(* unknown state *)
ELSE

	eState := E_TCPIP_IDLE;

	(* clear outputs *)
	bDone := FALSE;
	bBusy := FALSE;
	bError := FALSE;
	nErrorID := 0;
END_CASE

END_FUNCTION_BLOCK

// ---- POUs/SOFTWARE_lib/TCP FBs/FB_TCP_ReceiveData_V2.TcPOU
(* poll TCP Server for incoming data *)
FUNCTION_BLOCK FB_TCP_ReceiveData_V2
VAR_INPUT
	bEnable				: BOOL;			(* set TRUE to enable periodic TCP data receive *)
	hSocket				: T_HSocket;	(* TCP socket *)
	tUpdateTime			: TIME;			(* receive update rate *)
END_VAR
VAR_IN_OUT
	strTCPData			: T_MaxString;	(* string to which incoming TCP data will be appended *)
END_VAR
VAR_OUTPUT
	bDone				: BOOL;			(* TRUE = TCP receive done *)
	bBusy				: BOOL;			(* TRUE = TCP receive in progress *)
	bError				: BOOL;			(* TRUE = TCP receive error *)
	nErrorID			: UDINT;		(* TCP receive error code *)
	bDataReceived		: BOOL;			(* TRUE = data received *)
END_VAR
VAR
	fbTimer				: TON;
	eState				: E_TCPIP_State;
	fbTCPReceive		: FB_SocketReceive;
	strTCPRxChars		: T_MaxString;
END_VAR
(*
-------------------------------------------------------------------------------------------------
Date		Version	Author	Comments
-------------------------------------------------------------------------------------------------
16/08/2012	1.40.02	PB		Initial release

-------------------------------------------------------------------------------------------------
*)

(* TCP receive timer *)
fbTimer(
	IN	:= bEnable,
	PT	:= tUpdateTime
);

CASE eState OF

	(* idle state *)
	E_TCPIP_IDLE:

		(* receive data *)
		IF fbTimer.Q = TRUE THEN

			(* reset TCP receive timer *)
			fbTimer(IN := FALSE);

			(* update status outputs *)
			bDone := FALSE;
			bBusy := TRUE;
			bError := FALSE;
			nErrorID := 0;
			bDataReceived := FALSE;

			(* clear TCP receive string *)
			MEMSET(ADR(strTCPRxChars), 16#00, SIZEOF(strTCPRxChars));

			eState := E_TCPIP_RECEIVE;

		(* no action required *)
		ELSE

			bDone := FALSE;
			bBusy := FALSE;
			bError := FALSE;
			nErrorID := 0;
			bDataReceived := FALSE;
		END_IF


	(* receive data *)
	E_TCPIP_RECEIVE:

		(* receive data from TCP server *)
		fbTCPReceive(
			sSrvNetId	:= '',
			hSocket		:= hSocket,
			cbLen		:= SIZEOF(strTCPRxChars),
			pDest		:= ADR(strTCPRxChars),
			bExecute	:= TRUE,
			tTimeout	:= T#500ms
		);
		
		(* receive TCP data complete *)
		IF fbTCPReceive.bBusy = FALSE THEN
		
			(* receive TCP data completed OK *)
			IF fbTCPReceive.bError = FALSE THEN

				(* 1 or more data bytes received *)
				IF fbTCPReceive.nRecBytes > 0 THEN

					(* append returned data to TCP data string *)
					strTCPData := CONCAT(strTCPData, strTCPRxChars);
					bDataReceived := TRUE;

				(* no data received *)
				ELSE

					bDataReceived := FALSE;
				END_IF

			(* receive data error *)
			ELSE

				bError := TRUE;
				nErrorID := fbTCPReceive.nErrId;
			END_IF
		
			eState :=E_TCPIP_DONE;

			(* close off fbReceiveTCPData *)
			fbTCPReceive(bExecute := FALSE);
		END_IF


	(* done *)
	E_TCPIP_DONE:

		bDone := TRUE;
		bBusy := FALSE;

		eState :=E_TCPIP_IDLE;


	(* unknown state *)
	ELSE

		(* close off FBs *)
		fbTCPReceive(bExecute := FALSE);
		fbTimer(IN := FALSE);

		eState :=E_TCPIP_IDLE;

END_CASE

END_FUNCTION_BLOCK

// ---- POUs/SOFTWARE_lib/TCP FBs/FB_TCP_SendData.TcPOU
(* send data to TCP socket *)
FUNCTION_BLOCK FB_TCP_SendData
VAR_INPUT
	bExecute		: BOOL;			(* set TRUE to send data to TCP socket *)
	hSocket			: T_HSocket;	(* TCP socket handle *)
	pDataAdr		: POINTER TO BYTE;	(* pointer to data to send to TCP port *)
	nDataBytes		: UDINT;		(* number of bytes to send to TCP port *)
	tTimeout		: TIME;			(* TCP timeout *)
END_VAR
VAR_OUTPUT
	bDone			: BOOL;			(* TRUE = command complete *)
	bBusy			: BOOL;			(* TRUE = command in progress *)
	bError			: BOOL;			(* TRUE = error occurred with command *)
	nErrorID		: UDINT;		(* error code *)
END_VAR
VAR
	fbExecute		: R_TRIG;
	eState			: E_TCPIP_State;
	fbSendCommand	: FB_SocketSend;
END_VAR
(*
-------------------------------------------------------------------------------------------------
Date		Version	Author	Comments
-------------------------------------------------------------------------------------------------
			2.00.00	PB		Initial release

-------------------------------------------------------------------------------------------------
*)

(* compare files on rising edge of bExecute *)
fbExecute(CLK := bExecute);

CASE eState OF

	(* idle state *)
	E_TCPIP_IDLE:

		(* start new cycle *)
		IF fbExecute.Q = TRUE THEN

			(* reset status outputs *)
			bDone := FALSE;
			bBusy := TRUE;
			bError := FALSE;
			nErrorID := 0;

			eState := E_TCPIP_SEND;

		(* reset status outputs when bExecute is reset *)
		ELSIF bExecute = FALSE THEN

			bDone := FALSE;
			bBusy := FALSE;
			bError := FALSE;
			nErrorID := 0;
		END_IF


	(* send command *)
	E_TCPIP_SEND:

		(* send command *)
		fbSendCommand(
			sSrvNetId	:= '',
			hSocket		:= hSocket,
			cbLen		:= nDataBytes,
			pSrc		:= pDataAdr,
			bExecute	:= TRUE,
			tTimeout	:= T#1s,
		);

		(* send command complete *)
		IF fbSendCommand.bBusy = FALSE THEN

			(* send command completed OK *)
			IF fbSendCommand.bError = FALSE THEN

				eState := E_TCPIP_DONE;

			(* send command error *)
			ELSE

				bError := TRUE;
				nErrorID := fbSendCommand.nErrId;

				eState := E_TCPIP_DONE;
			END_IF

			(* close off fbSendCommand *)
			fbSendCommand(bExecute := FALSE);
		END_IF


	(* TCP command done *)
	E_TCPIP_DONE:

		bBusy := FALSE;
		bDone := TRUE;

		eState := E_TCPIP_IDLE;

(* unknown state *)
ELSE

	eState := E_TCPIP_IDLE;
END_CASE

END_FUNCTION_BLOCK

// ---- POUs/SOFTWARE_lib/TCP FBs/FB_TCP_ServerPortCtrl.TcPOU
(* TCP port ctrl for Server-Client devices *)
FUNCTION_BLOCK FB_TCP_ServerPortCtrl
VAR_INPUT
	bEnable				: BOOL;			(* set TRUE to enable TCP connection *)
	eMode				: E_SocketAcceptMode;	(* specifies which connections to accept *)
	strRemoteIPAddr		: T_IPv4Addr;	(* IP address for remote device *)
	strLocalIPAddr		: T_IPv4Addr;	(* IP address for local device *)
	nLocalPortNo		: UINT;			(* port number for local device *)
	tReconnectTime		: TIME;			(* TCP reconnect time *)
END_VAR
VAR_OUTPUT
	bConnected			: BOOL;			(* TRUE = TCP port is currently open *)
	bError				: BOOL;			(* TRUE = error occurred when opening TCP port *)
	nErrorID			: UDINT;		(* TRUE = error code *)
	hSocket				: T_HSocket;	(* TCP socket handle *)
	nSyncOffset			: DINT;			(* sync offset value to spread TCP Server access load *)
	eSocketState		: E_SocketConnectionState;	(* TCP socket state *)
END_VAR
VAR
	strTargetIPAddr		: T_IPv4Addr;
	arrTargetIPAddr		: T_IPv4AddrArr;
	nTargetPortNo		: UDINT;
	eTCPState			: E_TCPIP_State;
	bServerHndOK		: BOOL;
	hServer				: T_HSERVER;
	fbTCPPortCtrl		: FB_ServerClientConnection;
END_VAR
(*
-------------------------------------------------------------------------------------------------
Date		Version	Author	Comments
-------------------------------------------------------------------------------------------------
30/01/2015	3.00.00	PB		nRemotePort input removed as it is not used

-------------------------------------------------------------------------------------------------
06/09/2012	1.41.00	PB		FB now re-connects properly if strRemoteIPAddr or nRemotePortNo are changed while TCP connection is active.
							bError and nErrorID now linked directly to FB_ServerClientConnection.
22/11/2011	1.34.00	PB		Initial release.

-------------------------------------------------------------------------------------------------
*)

CASE eTCPState OF

	(* TCP connetion not active *)
	E_TCPIP_IDLE:

		(* TCP connection is enabled *)
		IF bEnable = TRUE THEN

			(* target IP address and port number *)
			strTargetIPAddr := strRemoteIPAddr;
			nTargetPortNo := nLocalPortNo;

			(* convert target IP address to bytes *)
			arrTargetIPAddr := F_ScanIPv4AddrIds(strTargetIPAddr);
			nSyncOffset := arrTargetIPAddr[3] MOD 10;

			eTCPState := E_TCPIP_CONNECT;
		END_IF


	(* open TCP connection *)
	E_TCPIP_CONNECT:

		(* close TCP connection *)
		IF bEnable = FALSE THEN

			eTCPState := E_TCPIP_DISCONNECT;

		(* TCP connect error or remote IP address or local port number have changed while connection is active *)
		ELSIF fbTCPPortCtrl.bError = TRUE OR (strRemoteIPAddr <> strTargetIPAddr AND strRemoteIPAddr <> '') OR (nLocalPortNo <> nTargetPortNo AND nLocalPortNo <> 0) THEN

			eTCPState := E_TCPIP_DISCONNECT;
		END_IF


	(* close TCP connection *)
	E_TCPIP_DISCONNECT:

		(* TCP port has been closed *)
		IF eSocketState = eSOCKET_DISCONNECTED THEN

			eTCPState := E_TCPIP_IDLE;
		END_IF


(* unknown state *)
ELSE

	eTCPState := E_TCPIP_IDLE;
END_CASE

(* create local server handle *)
bServerHndOK := F_CreateServerHnd('', strLocalIPAddr, nTargetPortNo, LISTEN_MODE_CLOSEALL(* OR CONNECT_MODE_ENABLEDBG*), FALSE, hServer);


(* TCP port connection ctrl *)
fbTCPPortCtrl(
	eMode		:= eMode,
	sRemoteHost	:= strTargetIPAddr,
	nRemotePort	:= nTargetPortNo,
	bEnable		:= bServerHndOK AND eTCPState = E_TCPIP_CONNECT,
	tReconnect	:= tReconnectTime,
	hServer		:= hServer,
	bError		=> bError,
	nErrID		=> nErrorID,
	hSocket		=> hSocket,
	eState		=> eSocketState
);

(* connected status *)
bConnected := eSocketState = eSOCKET_CONNECTED;

END_FUNCTION_BLOCK

// ---- POUs/Tests/FB_FIND_OuterDuplicates.TcPOU
FUNCTION_BLOCK FB_FIND_OuterDuplicates
VAR_INPUT
END_VAR
VAR_OUTPUT
	bHasDuplicates		: BOOL;
	nDuplicateCount		: UINT;
	nIterationCount		: UINT;
END_VAR
VAR
	nOuterIndex			: UINT;
	nMax_Outers			: UINT := 50;
	nMax_Packs			: UINT := 10;
	nInnerOuterIndex	: UINT;
	nInnerPackIndex		: UINT;
	nPackIndex			: UINT;
	sCurrentOuterCode	: T_MaxString;
	sCurrentPackCode	: T_MaxString;	
	bIsDuplicate 		: BOOL;
	bISOuterDuplicate	: BOOL;
END_VAR
VAR_IN_OUT	
	stCase				: ST_LAB_CaseData;
END_VAR


bHasDuplicates := FALSE;
nDuplicateCount := 0;
	
	(* Loop throught all packs in one case 'stCase' *)
	FOR nOuterIndex := 1 TO nMax_Outers DO
		sCurrentOuterCode := stCase.aOuters[nOuterIndex].sOuterCode;
		FOR nPackIndex := 1 TO nMax_Packs DO
			sCurrentPackCode := stCase.aOuters[nOuterIndex].aPacks[nPackIndex].sPackCode;
			bIsDuplicate := FALSE;			
			(* Looking for same pack codes in all outers *)
			FOR nInnerOuterIndex := nOuterIndex TO nMax_Outers DO
				IF nInnerOuterIndex < 50 THEN					
					IF (sCurrentOuterCode = stCase.aOuters[nInnerOuterIndex + 1].sOuterCode) THEN
						bIsOuterDuplicate									:= TRUE;													
						stCase.aOuters[nOuterIndex].nOuterRejectID			:= 200;					
						stCase.aOuters[nInnerOuterIndex + 1].nOuterRejectID	:= 200;
					END_IF	
				END_IF
				FOR nInnerPackIndex := 1 TO nMax_Packs DO
					nIterationCount	:= nIterationCount + 1;					
					(* Exclude comparing same pack with itself *)
					IF NOT ((nInnerOuterIndex = nOuterIndex) AND (nInnerPackIndex = nPackIndex)) THEN
						IF sCurrentPackCode = stCase.aOuters[nInnerOuterIndex].aPacks[nInnerPackIndex].sPackCode THEN
							bIsDuplicate := TRUE;
							nDuplicateCount := nDuplicateCount + 1;
							
							stCase.aOuters[nInnerOuterIndex].aPacks[nInnerPackIndex].nPackRejectID	:= 200;
							stCase.aOuters[nInnerOuterIndex].nOuterRejectID							:= 200;
							
							stCase.aOuters[nOuterIndex].aPacks[nPackIndex].nPackRejectID			:= 200;
							stCase.aOuters[nOuterIndex].nOuterRejectID								:= 200;
						END_IF
					END_IF
				END_FOR
			END_FOR			
			IF bIsDuplicate THEN
				bHasDuplicates 	:= TRUE;
			END_IF
		END_FOR
	END_FOR
	
	
	(* nDuplicateCount includes all elements with same pack codes *)
	(* the number of duplicated codes is nDuplicateCount/2 *)

END_FUNCTION_BLOCK

// ---- POUs/Tests/Outer_IN_Case_Duplicat.TcPOU
PROGRAM Outer_IN_Case_Duplicat
VAR
		
	fbFIND_OuterDuplicates		: FB_FIND_OuterDuplicates;
	
	bHasDuplicates				: BOOL;
	nDuplicateCount				: UINT;
	
	rTrig						: R_TRIG;
	bExecute					: BOOL;
	
	
	// dla petli for dla stworzenia outerow 
	rTrigDataFill	: R_TRIG;
	bDataFill		: BOOL;
	
	iOuter		: UINT;
	iPack		: UINT;
	
	sPackNum	: STRING;
	sOuterNum	: STRING;
	sPackCode	: STRING;
	
END_VAR


//CaseDataAdd();
//Case50outersADD();

FullFilOuter();

rTrig(CLK := bExecute);

IF rTrig.Q THEN	
	fbFIND_OuterDuplicates(
		stCase 			:= GVL_test.stCaseFull, 
		bHasDuplicates 	=> bHasDuplicates, 
		nDuplicateCount => nDuplicateCount
	);	
	
END_IF

ACTION Case50outersADD:
(* ===== OUTER 1 ===== *)
GVL_test.stCase.aOuters[1].sOuterCode    := 'OUTER1';
GVL_test.stCase.aOuters[1].nOutersStatus := 5;
// packs 1..10
GVL_test.stCase.aOuters[1].aPacks[1].sPackCode   := 'PACK01OUTER1';
GVL_test.stCase.aOuters[1].aPacks[1].nPackStatus := 5;
GVL_test.stCase.aOuters[1].aPacks[2].sPackCode   := 'PACK02OUTER1';
GVL_test.stCase.aOuters[1].aPacks[2].nPackStatus := 5;
GVL_test.stCase.aOuters[1].aPacks[3].sPackCode   := 'PACK03OUTER1';
GVL_test.stCase.aOuters[1].aPacks[3].nPackStatus := 5;
GVL_test.stCase.aOuters[1].aPacks[4].sPackCode   := 'PACK04OUTER1';
GVL_test.stCase.aOuters[1].aPacks[4].nPackStatus := 5;
GVL_test.stCase.aOuters[1].aPacks[5].sPackCode   := 'PACK05OUTER1';
GVL_test.stCase.aOuters[1].aPacks[5].nPackStatus := 5;
GVL_test.stCase.aOuters[1].aPacks[6].sPackCode   := 'PACK06OUTER1';
GVL_test.stCase.aOuters[1].aPacks[6].nPackStatus := 5;
GVL_test.stCase.aOuters[1].aPacks[7].sPackCode   := 'PACK07OUTER1';
GVL_test.stCase.aOuters[1].aPacks[7].nPackStatus := 5;
GVL_test.stCase.aOuters[1].aPacks[8].sPackCode   := 'PACK08OUTER1';
GVL_test.stCase.aOuters[1].aPacks[8].nPackStatus := 5;
GVL_test.stCase.aOuters[1].aPacks[9].sPackCode   := 'PACK09OUTER1';
GVL_test.stCase.aOuters[1].aPacks[9].nPackStatus := 5;
GVL_test.stCase.aOuters[1].aPacks[10].sPackCode  := 'PACK10OUTER1';
GVL_test.stCase.aOuters[1].aPacks[10].nPackStatus := 5;

(* ===== OUTER 2 ===== *)
GVL_test.stCase.aOuters[2].sOuterCode    := 'OUTER2';
GVL_test.stCase.aOuters[2].nOutersStatus := 5;
// packs 1..10
GVL_test.stCase.aOuters[2].aPacks[1].sPackCode   := 'PACK01OUTER2';
GVL_test.stCase.aOuters[2].aPacks[1].nPackStatus := 5;
GVL_test.stCase.aOuters[2].aPacks[2].sPackCode   := 'PACK02OUTER2';
GVL_test.stCase.aOuters[2].aPacks[2].nPackStatus := 5;
GVL_test.stCase.aOuters[2].aPacks[3].sPackCode   := 'PACK03OUTER2';
GVL_test.stCase.aOuters[2].aPacks[3].nPackStatus := 5;
GVL_test.stCase.aOuters[2].aPacks[4].sPackCode   := 'PACK04OUTER2';
GVL_test.stCase.aOuters[2].aPacks[4].nPackStatus := 5;
GVL_test.stCase.aOuters[2].aPacks[5].sPackCode   := 'PACK05OUTER2';
GVL_test.stCase.aOuters[2].aPacks[5].nPackStatus := 5;
GVL_test.stCase.aOuters[2].aPacks[6].sPackCode   := 'PACK06OUTER2';
GVL_test.stCase.aOuters[2].aPacks[6].nPackStatus := 5;
GVL_test.stCase.aOuters[2].aPacks[7].sPackCode   := 'PACK07OUTER2';
GVL_test.stCase.aOuters[2].aPacks[7].nPackStatus := 5;
GVL_test.stCase.aOuters[2].aPacks[8].sPackCode   := 'PACK08OUTER2';
GVL_test.stCase.aOuters[2].aPacks[8].nPackStatus := 5;
GVL_test.stCase.aOuters[2].aPacks[9].sPackCode   := 'PACK09OUTER2';
GVL_test.stCase.aOuters[2].aPacks[9].nPackStatus := 5;
GVL_test.stCase.aOuters[2].aPacks[10].sPackCode  := 'PACK10OUTER2';
GVL_test.stCase.aOuters[2].aPacks[10].nPackStatus := 5;

(* ===== OUTER 3 ===== *)
GVL_test.stCase.aOuters[3].sOuterCode    := 'OUTER3';
GVL_test.stCase.aOuters[3].nOutersStatus := 5;
// packs 1..10
GVL_test.stCase.aOuters[3].aPacks[1].sPackCode   := 'PACK01OUTER3';
GVL_test.stCase.aOuters[3].aPacks[1].nPackStatus := 5;
GVL_test.stCase.aOuters[3].aPacks[2].sPackCode   := 'PACK02OUTER3';
GVL_test.stCase.aOuters[3].aPacks[2].nPackStatus := 5;
GVL_test.stCase.aOuters[3].aPacks[3].sPackCode   := 'PACK03OUTER3';
GVL_test.stCase.aOuters[3].aPacks[3].nPackStatus := 5;
GVL_test.stCase.aOuters[3].aPacks[4].sPackCode   := 'PACK04OUTER3';
GVL_test.stCase.aOuters[3].aPacks[4].nPackStatus := 5;
GVL_test.stCase.aOuters[3].aPacks[5].sPackCode   := 'PACK05OUTER3';
GVL_test.stCase.aOuters[3].aPacks[5].nPackStatus := 5;
GVL_test.stCase.aOuters[3].aPacks[6].sPackCode   := 'PACK06OUTER3';
GVL_test.stCase.aOuters[3].aPacks[6].nPackStatus := 5;
GVL_test.stCase.aOuters[3].aPacks[7].sPackCode   := 'PACK07OUTER3';
GVL_test.stCase.aOuters[3].aPacks[7].nPackStatus := 5;
GVL_test.stCase.aOuters[3].aPacks[8].sPackCode   := 'PACK08OUTER3';
GVL_test.stCase.aOuters[3].aPacks[8].nPackStatus := 5;
GVL_test.stCase.aOuters[3].aPacks[9].sPackCode   := 'PACK09OUTER3';
GVL_test.stCase.aOuters[3].aPacks[9].nPackStatus := 5;
GVL_test.stCase.aOuters[3].aPacks[10].sPackCode  := 'PACK10OUTER3';
GVL_test.stCase.aOuters[3].aPacks[10].nPackStatus := 5;

(* ===== OUTER 4 ===== *)
GVL_test.stCase.aOuters[4].sOuterCode    := 'OUTER4';
GVL_test.stCase.aOuters[4].nOutersStatus := 5;
// packs 1..10
GVL_test.stCase.aOuters[4].aPacks[1].sPackCode   := 'PACK01OUTER4';
GVL_test.stCase.aOuters[4].aPacks[1].nPackStatus := 5;
GVL_test.stCase.aOuters[4].aPacks[2].sPackCode   := 'PACK02OUTER4';
GVL_test.stCase.aOuters[4].aPacks[2].nPackStatus := 5;
GVL_test.stCase.aOuters[4].aPacks[3].sPackCode   := 'PACK03OUTER4';
GVL_test.stCase.aOuters[4].aPacks[3].nPackStatus := 5;
GVL_test.stCase.aOuters[4].aPacks[4].sPackCode   := 'PACK04OUTER4';
GVL_test.stCase.aOuters[4].aPacks[4].nPackStatus := 5;
GVL_test.stCase.aOuters[4].aPacks[5].sPackCode   := 'PACK05OUTER4';
GVL_test.stCase.aOuters[4].aPacks[5].nPackStatus := 5;
GVL_test.stCase.aOuters[4].aPacks[6].sPackCode   := 'PACK06OUTER4';
GVL_test.stCase.aOuters[4].aPacks[6].nPackStatus := 5;
GVL_test.stCase.aOuters[4].aPacks[7].sPackCode   := 'PACK07OUTER4';
GVL_test.stCase.aOuters[4].aPacks[7].nPackStatus := 5;
GVL_test.stCase.aOuters[4].aPacks[8].sPackCode   := 'PACK08OUTER4';
GVL_test.stCase.aOuters[4].aPacks[8].nPackStatus := 5;
GVL_test.stCase.aOuters[4].aPacks[9].sPackCode   := 'PACK09OUTER4';
GVL_test.stCase.aOuters[4].aPacks[9].nPackStatus := 5;
GVL_test.stCase.aOuters[4].aPacks[10].sPackCode  := 'PACK10OUTER4';
GVL_test.stCase.aOuters[4].aPacks[10].nPackStatus := 5;

(* ===== OUTER 5 ===== *)
GVL_test.stCase.aOuters[5].sOuterCode    := 'OUTER5';
GVL_test.stCase.aOuters[5].nOutersStatus := 5;
// packs 1..10
GVL_test.stCase.aOuters[5].aPacks[1].sPackCode   := 'PACK01OUTER5';
GVL_test.stCase.aOuters[5].aPacks[1].nPackStatus := 5;
GVL_test.stCase.aOuters[5].aPacks[2].sPackCode   := 'PACK02OUTER5';
GVL_test.stCase.aOuters[5].aPacks[2].nPackStatus := 5;
GVL_test.stCase.aOuters[5].aPacks[3].sPackCode   := 'PACK03OUTER5';
GVL_test.stCase.aOuters[5].aPacks[3].nPackStatus := 5;
GVL_test.stCase.aOuters[5].aPacks[4].sPackCode   := 'PACK04OUTER5';
GVL_test.stCase.aOuters[5].aPacks[4].nPackStatus := 5;
GVL_test.stCase.aOuters[5].aPacks[5].sPackCode   := 'PACK05OUTER5';
GVL_test.stCase.aOuters[5].aPacks[5].nPackStatus := 5;
GVL_test.stCase.aOuters[5].aPacks[6].sPackCode   := 'PACK06OUTER5';
GVL_test.stCase.aOuters[5].aPacks[6].nPackStatus := 5;
GVL_test.stCase.aOuters[5].aPacks[7].sPackCode   := 'PACK07OUTER5';
GVL_test.stCase.aOuters[5].aPacks[7].nPackStatus := 5;
GVL_test.stCase.aOuters[5].aPacks[8].sPackCode   := 'PACK08OUTER5';
GVL_test.stCase.aOuters[5].aPacks[8].nPackStatus := 5;
GVL_test.stCase.aOuters[5].aPacks[9].sPackCode   := 'PACK09OUTER5';
GVL_test.stCase.aOuters[5].aPacks[9].nPackStatus := 5;
GVL_test.stCase.aOuters[5].aPacks[10].sPackCode  := 'PACK10OUTER5';
GVL_test.stCase.aOuters[5].aPacks[10].nPackStatus := 5;

(* ===== OUTER 6 ===== *)
GVL_test.stCase.aOuters[6].sOuterCode    := 'OUTER6';
GVL_test.stCase.aOuters[6].nOutersStatus := 5;
// packs 1..10
GVL_test.stCase.aOuters[6].aPacks[1].sPackCode   := 'PACK01OUTER6';
GVL_test.stCase.aOuters[6].aPacks[1].nPackStatus := 5;
GVL_test.stCase.aOuters[6].aPacks[2].sPackCode   := 'PACK02OUTER6';
GVL_test.stCase.aOuters[6].aPacks[2].nPackStatus := 5;
GVL_test.stCase.aOuters[6].aPacks[3].sPackCode   := 'PACK03OUTER6';
GVL_test.stCase.aOuters[6].aPacks[3].nPackStatus := 5;
GVL_test.stCase.aOuters[6].aPacks[4].sPackCode   := 'PACK04OUTER6';
GVL_test.stCase.aOuters[6].aPacks[4].nPackStatus := 5;
GVL_test.stCase.aOuters[6].aPacks[5].sPackCode   := 'PACK05OUTER6';
GVL_test.stCase.aOuters[6].aPacks[5].nPackStatus := 5;
GVL_test.stCase.aOuters[6].aPacks[6].sPackCode   := 'PACK06OUTER6';
GVL_test.stCase.aOuters[6].aPacks[6].nPackStatus := 5;
GVL_test.stCase.aOuters[6].aPacks[7].sPackCode   := 'PACK07OUTER6';
GVL_test.stCase.aOuters[6].aPacks[7].nPackStatus := 5;
GVL_test.stCase.aOuters[6].aPacks[8].sPackCode   := 'PACK08OUTER6';
GVL_test.stCase.aOuters[6].aPacks[8].nPackStatus := 5;
GVL_test.stCase.aOuters[6].aPacks[9].sPackCode   := 'PACK09OUTER6';
GVL_test.stCase.aOuters[6].aPacks[9].nPackStatus := 5;
GVL_test.stCase.aOuters[6].aPacks[10].sPackCode  := 'PACK10OUTER6';
GVL_test.stCase.aOuters[6].aPacks[10].nPackStatus := 5;

(* ===== OUTER 7 ===== *)
GVL_test.stCase.aOuters[7].sOuterCode    := 'OUTER7';
GVL_test.stCase.aOuters[7].nOutersStatus := 5;
// packs 1..10
GVL_test.stCase.aOuters[7].aPacks[1].sPackCode   := 'PACK01OUTER7';
GVL_test.stCase.aOuters[7].aPacks[1].nPackStatus := 5;
GVL_test.stCase.aOuters[7].aPacks[2].sPackCode   := 'PACK02OUTER7';
GVL_test.stCase.aOuters[7].aPacks[2].nPackStatus := 5;
GVL_test.stCase.aOuters[7].aPacks[3].sPackCode   := 'PACK03OUTER7';
GVL_test.stCase.aOuters[7].aPacks[3].nPackStatus := 5;
GVL_test.stCase.aOuters[7].aPacks[4].sPackCode   := 'PACK04OUTER7';
GVL_test.stCase.aOuters[7].aPacks[4].nPackStatus := 5;
GVL_test.stCase.aOuters[7].aPacks[5].sPackCode   := 'PACK05OUTER7';
GVL_test.stCase.aOuters[7].aPacks[5].nPackStatus := 5;
GVL_test.stCase.aOuters[7].aPacks[6].sPackCode   := 'PACK06OUTER7';
GVL_test.stCase.aOuters[7].aPacks[6].nPackStatus := 5;
GVL_test.stCase.aOuters[7].aPacks[7].sPackCode   := 'PACK07OUTER7';
GVL_test.stCase.aOuters[7].aPacks[7].nPackStatus := 5;
GVL_test.stCase.aOuters[7].aPacks[8].sPackCode   := 'PACK08OUTER7';
GVL_test.stCase.aOuters[7].aPacks[8].nPackStatus := 5;
GVL_test.stCase.aOuters[7].aPacks[9].sPackCode   := 'PACK09OUTER7';
GVL_test.stCase.aOuters[7].aPacks[9].nPackStatus := 5;
GVL_test.stCase.aOuters[7].aPacks[10].sPackCode  := 'PACK10OUTER7';
GVL_test.stCase.aOuters[7].aPacks[10].nPackStatus := 5;

(* ===== OUTER 8 ===== *)
GVL_test.stCase.aOuters[8].sOuterCode    := 'OUTER8';
GVL_test.stCase.aOuters[8].nOutersStatus := 5;
// packs 1..10
GVL_test.stCase.aOuters[8].aPacks[1].sPackCode   := 'PACK01OUTER8';
GVL_test.stCase.aOuters[8].aPacks[1].nPackStatus := 5;
GVL_test.stCase.aOuters[8].aPacks[2].sPackCode   := 'PACK02OUTER8';
GVL_test.stCase.aOuters[8].aPacks[2].nPackStatus := 5;
GVL_test.stCase.aOuters[8].aPacks[3].sPackCode   := 'PACK03OUTER8';
GVL_test.stCase.aOuters[8].aPacks[3].nPackStatus := 5;
GVL_test.stCase.aOuters[8].aPacks[4].sPackCode   := 'PACK04OUTER8';
GVL_test.stCase.aOuters[8].aPacks[4].nPackStatus := 5;
GVL_test.stCase.aOuters[8].aPacks[5].sPackCode   := 'PACK05OUTER8';
GVL_test.stCase.aOuters[8].aPacks[5].nPackStatus := 5;
GVL_test.stCase.aOuters[8].aPacks[6].sPackCode   := 'PACK06OUTER8';
GVL_test.stCase.aOuters[8].aPacks[6].nPackStatus := 5;
GVL_test.stCase.aOuters[8].aPacks[7].sPackCode   := 'PACK07OUTER8';
GVL_test.stCase.aOuters[8].aPacks[7].nPackStatus := 5;
GVL_test.stCase.aOuters[8].aPacks[8].sPackCode   := 'PACK08OUTER8';
GVL_test.stCase.aOuters[8].aPacks[8].nPackStatus := 5;
GVL_test.stCase.aOuters[8].aPacks[9].sPackCode   := 'PACK09OUTER8';
GVL_test.stCase.aOuters[8].aPacks[9].nPackStatus := 5;
GVL_test.stCase.aOuters[8].aPacks[10].sPackCode  := 'PACK10OUTER8';
GVL_test.stCase.aOuters[8].aPacks[10].nPackStatus := 5;

(* ===== OUTER 9 ===== *)
GVL_test.stCase.aOuters[9].sOuterCode    := 'OUTER9';
GVL_test.stCase.aOuters[9].nOutersStatus := 5;
// packs 1..10
GVL_test.stCase.aOuters[9].aPacks[1].sPackCode   := 'PACK01OUTER9';
GVL_test.stCase.aOuters[9].aPacks[1].nPackStatus := 5;
GVL_test.stCase.aOuters[9].aPacks[2].sPackCode   := 'PACK02OUTER9';
GVL_test.stCase.aOuters[9].aPacks[2].nPackStatus := 5;
GVL_test.stCase.aOuters[9].aPacks[3].sPackCode   := 'PACK03OUTER9';
GVL_test.stCase.aOuters[9].aPacks[3].nPackStatus := 5;
GVL_test.stCase.aOuters[9].aPacks[4].sPackCode   := 'PACK04OUTER9';
GVL_test.stCase.aOuters[9].aPacks[4].nPackStatus := 5;
GVL_test.stCase.aOuters[9].aPacks[5].sPackCode   := 'PACK05OUTER9';
GVL_test.stCase.aOuters[9].aPacks[5].nPackStatus := 5;
GVL_test.stCase.aOuters[9].aPacks[6].sPackCode   := 'PACK06OUTER9';
GVL_test.stCase.aOuters[9].aPacks[6].nPackStatus := 5;
GVL_test.stCase.aOuters[9].aPacks[7].sPackCode   := 'PACK07OUTER9';
GVL_test.stCase.aOuters[9].aPacks[7].nPackStatus := 5;
GVL_test.stCase.aOuters[9].aPacks[8].sPackCode   := 'PACK08OUTER9';
GVL_test.stCase.aOuters[9].aPacks[8].nPackStatus := 5;
GVL_test.stCase.aOuters[9].aPacks[9].sPackCode   := 'PACK09OUTER9';
GVL_test.stCase.aOuters[9].aPacks[9].nPackStatus := 5;
GVL_test.stCase.aOuters[9].aPacks[10].sPackCode  := 'PACK10OUTER9';
GVL_test.stCase.aOuters[9].aPacks[10].nPackStatus := 5;

(* ===== OUTER 10 ===== *)
GVL_test.stCase.aOuters[10].sOuterCode    := 'OUTER10';
GVL_test.stCase.aOuters[10].nOutersStatus := 5;
// packs 1..10
GVL_test.stCase.aOuters[10].aPacks[1].sPackCode   := 'PACK01OUTER10';
GVL_test.stCase.aOuters[10].aPacks[1].nPackStatus := 5;
GVL_test.stCase.aOuters[10].aPacks[2].sPackCode   := 'PACK02OUTER10';
GVL_test.stCase.aOuters[10].aPacks[2].nPackStatus := 5;
GVL_test.stCase.aOuters[10].aPacks[3].sPackCode   := 'PACK03OUTER10';
GVL_test.stCase.aOuters[10].aPacks[3].nPackStatus := 5;
GVL_test.stCase.aOuters[10].aPacks[4].sPackCode   := 'PACK04OUTER10';
GVL_test.stCase.aOuters[10].aPacks[4].nPackStatus := 5;
GVL_test.stCase.aOuters[10].aPacks[5].sPackCode   := 'PACK05OUTER10';
GVL_test.stCase.aOuters[10].aPacks[5].nPackStatus := 5;
GVL_test.stCase.aOuters[10].aPacks[6].sPackCode   := 'PACK06OUTER10';
GVL_test.stCase.aOuters[10].aPacks[6].nPackStatus := 5;
GVL_test.stCase.aOuters[10].aPacks[7].sPackCode   := 'PACK07OUTER10';
GVL_test.stCase.aOuters[10].aPacks[7].nPackStatus := 5;
GVL_test.stCase.aOuters[10].aPacks[8].sPackCode   := 'PACK08OUTER10';
GVL_test.stCase.aOuters[10].aPacks[8].nPackStatus := 5;
GVL_test.stCase.aOuters[10].aPacks[9].sPackCode   := 'PACK09OUTER10';
GVL_test.stCase.aOuters[10].aPacks[9].nPackStatus := 5;
GVL_test.stCase.aOuters[10].aPacks[10].sPackCode  := 'PACK10OUTER10';
GVL_test.stCase.aOuters[10].aPacks[10].nPackStatus := 5;
////////////////////////////////////////////////////////////////////////////////////
(* ===== OUTER 11 ===== *)
GVL_test.stCase.aOuters[11].sOuterCode    := 'OUTER1';
GVL_test.stCase.aOuters[11].nOutersStatus := 5;
// packs 1..10
GVL_test.stCase.aOuters[11].aPacks[1].sPackCode   := 'PACK01OUTER11';
GVL_test.stCase.aOuters[11].aPacks[1].nPackStatus := 5;
GVL_test.stCase.aOuters[11].aPacks[2].sPackCode   := 'PACK02OUTER11';
GVL_test.stCase.aOuters[11].aPacks[2].nPackStatus := 5;
GVL_test.stCase.aOuters[11].aPacks[3].sPackCode   := 'PACK03OUTER11';
GVL_test.stCase.aOuters[11].aPacks[3].nPackStatus := 5;
GVL_test.stCase.aOuters[11].aPacks[4].sPackCode   := 'PACK04OUTER11';
GVL_test.stCase.aOuters[11].aPacks[4].nPackStatus := 5;
GVL_test.stCase.aOuters[11].aPacks[5].sPackCode   := 'PACK05OUTER11';
GVL_test.stCase.aOuters[11].aPacks[5].nPackStatus := 5;
GVL_test.stCase.aOuters[11].aPacks[6].sPackCode   := 'PACK06OUTER11';
GVL_test.stCase.aOuters[11].aPacks[6].nPackStatus := 5;
GVL_test.stCase.aOuters[11].aPacks[7].sPackCode   := 'PACK07OUTER11';
GVL_test.stCase.aOuters[11].aPacks[7].nPackStatus := 5;
GVL_test.stCase.aOuters[11].aPacks[8].sPackCode   := 'PACK08OUTER11';
GVL_test.stCase.aOuters[11].aPacks[8].nPackStatus := 5;
GVL_test.stCase.aOuters[11].aPacks[9].sPackCode   := 'PACK09OUTER11';
GVL_test.stCase.aOuters[11].aPacks[9].nPackStatus := 5;
GVL_test.stCase.aOuters[11].aPacks[10].sPackCode  := 'PACK10OUTER11';
GVL_test.stCase.aOuters[11].aPacks[10].nPackStatus := 5;

(* ===== OUTER 12 ===== *)
GVL_test.stCase.aOuters[12].sOuterCode    := 'OUTER2';
GVL_test.stCase.aOuters[12].nOutersStatus := 5;
// packs 1..10
GVL_test.stCase.aOuters[12].aPacks[1].sPackCode   := 'PACK01OUTER12';
GVL_test.stCase.aOuters[12].aPacks[1].nPackStatus := 5;
GVL_test.stCase.aOuters[12].aPacks[2].sPackCode   := 'PACK02OUTER12';
GVL_test.stCase.aOuters[12].aPacks[2].nPackStatus := 5;
GVL_test.stCase.aOuters[12].aPacks[3].sPackCode   := 'PACK03OUTER12';
GVL_test.stCase.aOuters[12].aPacks[3].nPackStatus := 5;
GVL_test.stCase.aOuters[12].aPacks[4].sPackCode   := 'PACK04OUTER12';
GVL_test.stCase.aOuters[12].aPacks[4].nPackStatus := 5;
GVL_test.stCase.aOuters[12].aPacks[5].sPackCode   := 'PACK05OUTER12';
GVL_test.stCase.aOuters[12].aPacks[5].nPackStatus := 5;
GVL_test.stCase.aOuters[12].aPacks[6].sPackCode   := 'PACK06OUTER12';
GVL_test.stCase.aOuters[12].aPacks[6].nPackStatus := 5;
GVL_test.stCase.aOuters[12].aPacks[7].sPackCode   := 'PACK07OUTER12';
GVL_test.stCase.aOuters[12].aPacks[7].nPackStatus := 5;
GVL_test.stCase.aOuters[12].aPacks[8].sPackCode   := 'PACK08OUTER12';
GVL_test.stCase.aOuters[12].aPacks[8].nPackStatus := 5;
GVL_test.stCase.aOuters[12].aPacks[9].sPackCode   := 'PACK09OUTER12';
GVL_test.stCase.aOuters[12].aPacks[9].nPackStatus := 5;
GVL_test.stCase.aOuters[12].aPacks[10].sPackCode  := 'PACK10OUTER12';
GVL_test.stCase.aOuters[12].aPacks[10].nPackStatus := 5;

(* ===== OUTER 3 ===== *)
GVL_test.stCase.aOuters[3].sOuterCode    := 'OUTER3';
GVL_test.stCase.aOuters[3].nOutersStatus := 5;
// packs 1..10
GVL_test.stCase.aOuters[3].aPacks[1].sPackCode   := 'PACK01OUTER3';
GVL_test.stCase.aOuters[3].aPacks[1].nPackStatus := 5;
GVL_test.stCase.aOuters[3].aPacks[2].sPackCode   := 'PACK02OUTER3';
GVL_test.stCase.aOuters[3].aPacks[2].nPackStatus := 5;
GVL_test.stCase.aOuters[3].aPacks[3].sPackCode   := 'PACK03OUTER3';
GVL_test.stCase.aOuters[3].aPacks[3].nPackStatus := 5;
GVL_test.stCase.aOuters[3].aPacks[4].sPackCode   := 'PACK04OUTER3';
GVL_test.stCase.aOuters[3].aPacks[4].nPackStatus := 5;
GVL_test.stCase.aOuters[3].aPacks[5].sPackCode   := 'PACK05OUTER3';
GVL_test.stCase.aOuters[3].aPacks[5].nPackStatus := 5;
GVL_test.stCase.aOuters[3].aPacks[6].sPackCode   := 'PACK06OUTER3';
GVL_test.stCase.aOuters[3].aPacks[6].nPackStatus := 5;
GVL_test.stCase.aOuters[3].aPacks[7].sPackCode   := 'PACK07OUTER3';
GVL_test.stCase.aOuters[3].aPacks[7].nPackStatus := 5;
GVL_test.stCase.aOuters[3].aPacks[8].sPackCode   := 'PACK08OUTER3';
GVL_test.stCase.aOuters[3].aPacks[8].nPackStatus := 5;
GVL_test.stCase.aOuters[3].aPacks[9].sPackCode   := 'PACK09OUTER3';
GVL_test.stCase.aOuters[3].aPacks[9].nPackStatus := 5;
GVL_test.stCase.aOuters[3].aPacks[10].sPackCode  := 'PACK10OUTER3';
GVL_test.stCase.aOuters[3].aPacks[10].nPackStatus := 5;

(* ===== OUTER 4 ===== *)
GVL_test.stCase.aOuters[4].sOuterCode    := 'OUTER4';
GVL_test.stCase.aOuters[4].nOutersStatus := 5;
// packs 1..10
GVL_test.stCase.aOuters[4].aPacks[1].sPackCode   := 'PACK01OUTER4';
GVL_test.stCase.aOuters[4].aPacks[1].nPackStatus := 5;
GVL_test.stCase.aOuters[4].aPacks[2].sPackCode   := 'PACK02OUTER4';
GVL_test.stCase.aOuters[4].aPacks[2].nPackStatus := 5;
GVL_test.stCase.aOuters[4].aPacks[3].sPackCode   := 'PACK03OUTER4';
GVL_test.stCase.aOuters[4].aPacks[3].nPackStatus := 5;
GVL_test.stCase.aOuters[4].aPacks[4].sPackCode   := 'PACK04OUTER4';
GVL_test.stCase.aOuters[4].aPacks[4].nPackStatus := 5;
GVL_test.stCase.aOuters[4].aPacks[5].sPackCode   := 'PACK05OUTER4';
GVL_test.stCase.aOuters[4].aPacks[5].nPackStatus := 5;
GVL_test.stCase.aOuters[4].aPacks[6].sPackCode   := 'PACK06OUTER4';
GVL_test.stCase.aOuters[4].aPacks[6].nPackStatus := 5;
GVL_test.stCase.aOuters[4].aPacks[7].sPackCode   := 'PACK07OUTER4';
GVL_test.stCase.aOuters[4].aPacks[7].nPackStatus := 5;
GVL_test.stCase.aOuters[4].aPacks[8].sPackCode   := 'PACK08OUTER4';
GVL_test.stCase.aOuters[4].aPacks[8].nPackStatus := 5;
GVL_test.stCase.aOuters[4].aPacks[9].sPackCode   := 'PACK09OUTER4';
GVL_test.stCase.aOuters[4].aPacks[9].nPackStatus := 5;
GVL_test.stCase.aOuters[4].aPacks[10].sPackCode  := 'PACK10OUTER4';
GVL_test.stCase.aOuters[4].aPacks[10].nPackStatus := 5;

(* ===== OUTER 5 ===== *)
GVL_test.stCase.aOuters[5].sOuterCode    := 'OUTER5';
GVL_test.stCase.aOuters[5].nOutersStatus := 5;
// packs 1..10
GVL_test.stCase.aOuters[5].aPacks[1].sPackCode   := 'PACK01OUTER5';
GVL_test.stCase.aOuters[5].aPacks[1].nPackStatus := 5;
GVL_test.stCase.aOuters[5].aPacks[2].sPackCode   := 'PACK02OUTER5';
GVL_test.stCase.aOuters[5].aPacks[2].nPackStatus := 5;
GVL_test.stCase.aOuters[5].aPacks[3].sPackCode   := 'PACK03OUTER5';
GVL_test.stCase.aOuters[5].aPacks[3].nPackStatus := 5;
GVL_test.stCase.aOuters[5].aPacks[4].sPackCode   := 'PACK04OUTER5';
GVL_test.stCase.aOuters[5].aPacks[4].nPackStatus := 5;
GVL_test.stCase.aOuters[5].aPacks[5].sPackCode   := 'PACK05OUTER5';
GVL_test.stCase.aOuters[5].aPacks[5].nPackStatus := 5;
GVL_test.stCase.aOuters[5].aPacks[6].sPackCode   := 'PACK06OUTER5';
GVL_test.stCase.aOuters[5].aPacks[6].nPackStatus := 5;
GVL_test.stCase.aOuters[5].aPacks[7].sPackCode   := 'PACK07OUTER5';
GVL_test.stCase.aOuters[5].aPacks[7].nPackStatus := 5;
GVL_test.stCase.aOuters[5].aPacks[8].sPackCode   := 'PACK08OUTER5';
GVL_test.stCase.aOuters[5].aPacks[8].nPackStatus := 5;
GVL_test.stCase.aOuters[5].aPacks[9].sPackCode   := 'PACK09OUTER5';
GVL_test.stCase.aOuters[5].aPacks[9].nPackStatus := 5;
GVL_test.stCase.aOuters[5].aPacks[10].sPackCode  := 'PACK10OUTER5';
GVL_test.stCase.aOuters[5].aPacks[10].nPackStatus := 5;

(* ===== OUTER 6 ===== *)
GVL_test.stCase.aOuters[6].sOuterCode    := 'OUTER6';
GVL_test.stCase.aOuters[6].nOutersStatus := 5;
// packs 1..10
GVL_test.stCase.aOuters[6].aPacks[1].sPackCode   := 'PACK01OUTER6';
GVL_test.stCase.aOuters[6].aPacks[1].nPackStatus := 5;
GVL_test.stCase.aOuters[6].aPacks[2].sPackCode   := 'PACK02OUTER6';
GVL_test.stCase.aOuters[6].aPacks[2].nPackStatus := 5;
GVL_test.stCase.aOuters[6].aPacks[3].sPackCode   := 'PACK03OUTER6';
GVL_test.stCase.aOuters[6].aPacks[3].nPackStatus := 5;
GVL_test.stCase.aOuters[6].aPacks[4].sPackCode   := 'PACK04OUTER6';
GVL_test.stCase.aOuters[6].aPacks[4].nPackStatus := 5;
GVL_test.stCase.aOuters[6].aPacks[5].sPackCode   := 'PACK05OUTER6';
GVL_test.stCase.aOuters[6].aPacks[5].nPackStatus := 5;
GVL_test.stCase.aOuters[6].aPacks[6].sPackCode   := 'PACK06OUTER6';
GVL_test.stCase.aOuters[6].aPacks[6].nPackStatus := 5;
GVL_test.stCase.aOuters[6].aPacks[7].sPackCode   := 'PACK07OUTER6';
GVL_test.stCase.aOuters[6].aPacks[7].nPackStatus := 5;
GVL_test.stCase.aOuters[6].aPacks[8].sPackCode   := 'PACK08OUTER6';
GVL_test.stCase.aOuters[6].aPacks[8].nPackStatus := 5;
GVL_test.stCase.aOuters[6].aPacks[9].sPackCode   := 'PACK09OUTER6';
GVL_test.stCase.aOuters[6].aPacks[9].nPackStatus := 5;
GVL_test.stCase.aOuters[6].aPacks[10].sPackCode  := 'PACK10OUTER6';
GVL_test.stCase.aOuters[6].aPacks[10].nPackStatus := 5;

(* ===== OUTER 7 ===== *)
GVL_test.stCase.aOuters[7].sOuterCode    := 'OUTER7';
GVL_test.stCase.aOuters[7].nOutersStatus := 5;
// packs 1..10
GVL_test.stCase.aOuters[7].aPacks[1].sPackCode   := 'PACK01OUTER7';
GVL_test.stCase.aOuters[7].aPacks[1].nPackStatus := 5;
GVL_test.stCase.aOuters[7].aPacks[2].sPackCode   := 'PACK02OUTER7';
GVL_test.stCase.aOuters[7].aPacks[2].nPackStatus := 5;
GVL_test.stCase.aOuters[7].aPacks[3].sPackCode   := 'PACK03OUTER7';
GVL_test.stCase.aOuters[7].aPacks[3].nPackStatus := 5;
GVL_test.stCase.aOuters[7].aPacks[4].sPackCode   := 'PACK04OUTER7';
GVL_test.stCase.aOuters[7].aPacks[4].nPackStatus := 5;
GVL_test.stCase.aOuters[7].aPacks[5].sPackCode   := 'PACK05OUTER7';
GVL_test.stCase.aOuters[7].aPacks[5].nPackStatus := 5;
GVL_test.stCase.aOuters[7].aPacks[6].sPackCode   := 'PACK06OUTER7';
GVL_test.stCase.aOuters[7].aPacks[6].nPackStatus := 5;
GVL_test.stCase.aOuters[7].aPacks[7].sPackCode   := 'PACK07OUTER7';
GVL_test.stCase.aOuters[7].aPacks[7].nPackStatus := 5;
GVL_test.stCase.aOuters[7].aPacks[8].sPackCode   := 'PACK08OUTER7';
GVL_test.stCase.aOuters[7].aPacks[8].nPackStatus := 5;
GVL_test.stCase.aOuters[7].aPacks[9].sPackCode   := 'PACK09OUTER7';
GVL_test.stCase.aOuters[7].aPacks[9].nPackStatus := 5;
GVL_test.stCase.aOuters[7].aPacks[10].sPackCode  := 'PACK10OUTER7';
GVL_test.stCase.aOuters[7].aPacks[10].nPackStatus := 5;

(* ===== OUTER 8 ===== *)
GVL_test.stCase.aOuters[8].sOuterCode    := 'OUTER8';
GVL_test.stCase.aOuters[8].nOutersStatus := 5;
// packs 1..10
GVL_test.stCase.aOuters[8].aPacks[1].sPackCode   := 'PACK01OUTER8';
GVL_test.stCase.aOuters[8].aPacks[1].nPackStatus := 5;
GVL_test.stCase.aOuters[8].aPacks[2].sPackCode   := 'PACK02OUTER8';
GVL_test.stCase.aOuters[8].aPacks[2].nPackStatus := 5;
GVL_test.stCase.aOuters[8].aPacks[3].sPackCode   := 'PACK03OUTER8';
GVL_test.stCase.aOuters[8].aPacks[3].nPackStatus := 5;
GVL_test.stCase.aOuters[8].aPacks[4].sPackCode   := 'PACK04OUTER8';
GVL_test.stCase.aOuters[8].aPacks[4].nPackStatus := 5;
GVL_test.stCase.aOuters[8].aPacks[5].sPackCode   := 'PACK05OUTER8';
GVL_test.stCase.aOuters[8].aPacks[5].nPackStatus := 5;
GVL_test.stCase.aOuters[8].aPacks[6].sPackCode   := 'PACK06OUTER8';
GVL_test.stCase.aOuters[8].aPacks[6].nPackStatus := 5;
GVL_test.stCase.aOuters[8].aPacks[7].sPackCode   := 'PACK07OUTER8';
GVL_test.stCase.aOuters[8].aPacks[7].nPackStatus := 5;
GVL_test.stCase.aOuters[8].aPacks[8].sPackCode   := 'PACK08OUTER8';
GVL_test.stCase.aOuters[8].aPacks[8].nPackStatus := 5;
GVL_test.stCase.aOuters[8].aPacks[9].sPackCode   := 'PACK09OUTER8';
GVL_test.stCase.aOuters[8].aPacks[9].nPackStatus := 5;
GVL_test.stCase.aOuters[8].aPacks[10].sPackCode  := 'PACK10OUTER8';
GVL_test.stCase.aOuters[8].aPacks[10].nPackStatus := 5;

(* ===== OUTER 9 ===== *)
GVL_test.stCase.aOuters[9].sOuterCode    := 'OUTER9';
GVL_test.stCase.aOuters[9].nOutersStatus := 5;
// packs 1..10
GVL_test.stCase.aOuters[9].aPacks[1].sPackCode   := 'PACK01OUTER9';
GVL_test.stCase.aOuters[9].aPacks[1].nPackStatus := 5;
GVL_test.stCase.aOuters[9].aPacks[2].sPackCode   := 'PACK02OUTER9';
GVL_test.stCase.aOuters[9].aPacks[2].nPackStatus := 5;
GVL_test.stCase.aOuters[9].aPacks[3].sPackCode   := 'PACK03OUTER9';
GVL_test.stCase.aOuters[9].aPacks[3].nPackStatus := 5;
GVL_test.stCase.aOuters[9].aPacks[4].sPackCode   := 'PACK04OUTER9';
GVL_test.stCase.aOuters[9].aPacks[4].nPackStatus := 5;
GVL_test.stCase.aOuters[9].aPacks[5].sPackCode   := 'PACK05OUTER9';
GVL_test.stCase.aOuters[9].aPacks[5].nPackStatus := 5;
GVL_test.stCase.aOuters[9].aPacks[6].sPackCode   := 'PACK06OUTER9';
GVL_test.stCase.aOuters[9].aPacks[6].nPackStatus := 5;
GVL_test.stCase.aOuters[9].aPacks[7].sPackCode   := 'PACK07OUTER9';
GVL_test.stCase.aOuters[9].aPacks[7].nPackStatus := 5;
GVL_test.stCase.aOuters[9].aPacks[8].sPackCode   := 'PACK08OUTER9';
GVL_test.stCase.aOuters[9].aPacks[8].nPackStatus := 5;
GVL_test.stCase.aOuters[9].aPacks[9].sPackCode   := 'PACK09OUTER9';
GVL_test.stCase.aOuters[9].aPacks[9].nPackStatus := 5;
GVL_test.stCase.aOuters[9].aPacks[10].sPackCode  := 'PACK10OUTER9';
GVL_test.stCase.aOuters[9].aPacks[10].nPackStatus := 5;

(* ===== OUTER 10 ===== *)
GVL_test.stCase.aOuters[10].sOuterCode    := 'OUTER10';
GVL_test.stCase.aOuters[10].nOutersStatus := 5;
// packs 1..10
GVL_test.stCase.aOuters[10].aPacks[1].sPackCode   := 'PACK01OUTER10';
GVL_test.stCase.aOuters[10].aPacks[1].nPackStatus := 5;
GVL_test.stCase.aOuters[10].aPacks[2].sPackCode   := 'PACK02OUTER10';
GVL_test.stCase.aOuters[10].aPacks[2].nPackStatus := 5;
GVL_test.stCase.aOuters[10].aPacks[3].sPackCode   := 'PACK03OUTER10';
GVL_test.stCase.aOuters[10].aPacks[3].nPackStatus := 5;
GVL_test.stCase.aOuters[10].aPacks[4].sPackCode   := 'PACK04OUTER10';
GVL_test.stCase.aOuters[10].aPacks[4].nPackStatus := 5;
GVL_test.stCase.aOuters[10].aPacks[5].sPackCode   := 'PACK05OUTER10';
GVL_test.stCase.aOuters[10].aPacks[5].nPackStatus := 5;
GVL_test.stCase.aOuters[10].aPacks[6].sPackCode   := 'PACK06OUTER10';
GVL_test.stCase.aOuters[10].aPacks[6].nPackStatus := 5;
GVL_test.stCase.aOuters[10].aPacks[7].sPackCode   := 'PACK07OUTER10';
GVL_test.stCase.aOuters[10].aPacks[7].nPackStatus := 5;
GVL_test.stCase.aOuters[10].aPacks[8].sPackCode   := 'PACK08OUTER10';
GVL_test.stCase.aOuters[10].aPacks[8].nPackStatus := 5;
GVL_test.stCase.aOuters[10].aPacks[9].sPackCode   := 'PACK09OUTER10';
GVL_test.stCase.aOuters[10].aPacks[9].nPackStatus := 5;
GVL_test.stCase.aOuters[10].aPacks[10].sPackCode  := 'PACK10OUTER10';
GVL_test.stCase.aOuters[10].aPacks[10].nPackStatus := 5;
END_ACTION

ACTION CaseDataAdd:
(*     outer 1 data     *)
GVL_test.stCase.aOuters[1].sOuterCode 	:= 'OUTER1';
GVL_test.stCase.aOuters[1].nOutersStatus	:= 5;
// packs 1..10
GVL_test.stCase.aOuters[1].aPacks[1].sPackCode 		:= 'PACK01OUTER1';
GVL_test.stCase.aOuters[1].aPacks[1].nPackStatus 	:= 5;
GVL_test.stCase.aOuters[1].aPacks[2].sPackCode 		:= 'PACK02OUTER1';
GVL_test.stCase.aOuters[1].aPacks[2].nPackStatus 	:= 5;
GVL_test.stCase.aOuters[1].aPacks[3].sPackCode 		:= 'PACK03OUTER1';
GVL_test.stCase.aOuters[1].aPacks[3].nPackStatus 	:= 5;
GVL_test.stCase.aOuters[1].aPacks[4].sPackCode 		:= 'PACK04OUTER1';
GVL_test.stCase.aOuters[1].aPacks[4].nPackStatus 	:= 5;
GVL_test.stCase.aOuters[1].aPacks[5].sPackCode 		:= 'PACK05OUTER1';
GVL_test.stCase.aOuters[1].aPacks[5].nPackStatus 	:= 5;
GVL_test.stCase.aOuters[1].aPacks[6].sPackCode 		:= 'PACK06OUTER1';
GVL_test.stCase.aOuters[1].aPacks[6].nPackStatus 	:= 5;
GVL_test.stCase.aOuters[1].aPacks[7].sPackCode 		:= 'PACK07OUTER1';
GVL_test.stCase.aOuters[1].aPacks[7].nPackStatus 	:= 5;
GVL_test.stCase.aOuters[1].aPacks[8].sPackCode 		:= 'PACK08OUTER1';
GVL_test.stCase.aOuters[1].aPacks[8].nPackStatus 	:= 5;
GVL_test.stCase.aOuters[1].aPacks[9].sPackCode 		:= 'PACK09OUTER1';
GVL_test.stCase.aOuters[1].aPacks[9].nPackStatus 	:= 5;
GVL_test.stCase.aOuters[1].aPacks[10].sPackCode 	:= 'PACK10OUTER1';
GVL_test.stCase.aOuters[1].aPacks[10].nPackStatus 	:= 5;



(*     outer 1 data     *)
GVL_test.stCase.aOuters[2].sOuterCode 	:= 'OUTER1';
GVL_test.stCase.aOuters[2].nOutersStatus	:= 5;
// packs 1 data
GVL_test.stCase.aOuters[2].aPacks[1].sPackCode 	:= 'PACK01OUTER1';
GVL_test.stCase.aOuters[2].aPacks[1].nPackStatus := 5;
// packs 2 data
GVL_test.stCase.aOuters[2].aPacks[2].sPackCode 	:= 'PACK02OUTER1';
GVL_test.stCase.aOuters[2].aPacks[2].nPackStatus := 5;
// packs 3 data
GVL_test.stCase.aOuters[2].aPacks[3].sPackCode 	:= 'PACK03OUTER1';
GVL_test.stCase.aOuters[2].aPacks[3].nPackStatus := 5;

(*     outer 2 data     *)
GVL_test.stCase.aOuters[2].sOuterCode 	:= 'OUTER2';
GVL_test.stCase.aOuters[2].nOutersStatus	:= 5;
// packs 1 data
GVL_test.stCase.aOuters[2].aPacks[1].sPackCode 	:= 'PACK01OUTER2';
GVL_test.stCase.aOuters[2].aPacks[1].nPackStatus := 5;
// packs 2 data
GVL_test.stCase.aOuters[2].aPacks[2].sPackCode 	:= 'PACK02OUTER2';
GVL_test.stCase.aOuters[2].aPacks[2].nPackStatus := 5;
// packs 3 data
GVL_test.stCase.aOuters[2].aPacks[3].sPackCode 	:= 'PACK03OUTER2';
GVL_test.stCase.aOuters[2].aPacks[3].nPackStatus := 5;


(*     outer 3 data     *)
GVL_test.stCase.aOuters[3].sOuterCode 	:= 'OUTER3';
GVL_test.stCase.aOuters[3].nOutersStatus	:= 5;
// packs 1 data
GVL_test.stCase.aOuters[3].aPacks[1].sPackCode 	:= 'PACK01OUTER3';
GVL_test.stCase.aOuters[3].aPacks[1].nPackStatus := 5;
// packs 2 data
GVL_test.stCase.aOuters[3].aPacks[2].sPackCode 	:= 'PACK02OUTER3';
GVL_test.stCase.aOuters[3].aPacks[2].nPackStatus := 5;
// packs 3 data
GVL_test.stCase.aOuters[3].aPacks[3].sPackCode 	:= 'PACK03OUTER3';
GVL_test.stCase.aOuters[3].aPacks[3].nPackStatus := 5;
END_ACTION

ACTION FullFilOuter:

rTrigDataFill(CLK := bDataFill);

IF rTrigDataFill.Q THEN
	
	FOR iOuter := 1 TO 50 DO
		(* Ustaw outer *)
		GVL_test.stCaseFull.aOuters[iOuter].sOuterCode    := CONCAT('OUTER', INT_TO_STRING(iOuter));
		GVL_test.stCaseFull.aOuters[iOuter].nOutersStatus := 5;
		
		FOR iPack := 1 TO 10 DO
			(* Pack number z zerami *)
			sPackNum := CONCAT('0', INT_TO_STRING(iPack));  (* dla 1-9: '01'-'09' *)
			IF iPack = 10 THEN
				sPackNum := '10';
			END_IF;
			
			(* Outer number z zerami dla 1-9 *)
			sOuterNum := CONCAT('0', INT_TO_STRING(iOuter));
			IF iOuter >= 10 THEN
				sOuterNum := INT_TO_STRING(iOuter);
			END_IF;
			
			(* Sklej pack code *)
			sPackCode := CONCAT(CONCAT('PACK', sPackNum), CONCAT('OUTER', sOuterNum));
			
			(* Przypisz *)
			GVL_test.stCaseFull.aOuters[iOuter].aPacks[iPack].sPackCode   := sPackCode;
			GVL_test.stCaseFull.aOuters[iOuter].aPacks[iPack].nPackStatus := 5;
		END_FOR;
	END_FOR;
	
END_IF
END_ACTION

END_PROGRAM

// ---- POUs/Tests/PRG_Test.TcPOU
PROGRAM PRG_Test
VAR
	nMaxBytes: UDINT;
	strTCPRxString: STRING(255);
	
	strTargetIPAddr		: T_IPv4Addr := '192.168.1.44';	
	arrTargetIPAddr		: T_IPv4AddrArr;
	nSyncOffset			: DINT;		
	nSyncOffset_1		: DINT;	
	tTaskTime			: TIME := T#200MS;
	sString_1			: STRING(255);
	sString_2			: STRING(255);
	sConcuted			: STRING(1023);
	bConcuted			: BOOL;
	
	nSize_1				: UINT;
	nSize_2				: UINT;
	nSize_3				: UDINT;
	nStatusByte			: BYTE;
	bitNO				: USINT := 6;
	nBytesQuantity		: INT :=1;
	nBytePosition		: INT :=5;
	sString_4			: STRING(255);
	strTCPRxDebug		: ARRAY[1..20] OF  STRING(100);
	nSizeTCPRxDebug		: UINT;
	sStringTest			: STRING(100) := '_STRING_W_PIERWSZEJ_TABLICY_';
	nIndex				: INT;
	nSizeTCPRxDebug_1	: UINT;
END_VAR


nMaxBytes := SIZEOF(strTCPRxString) - INT_TO_UDINT(LEN(strTCPRxString) - 1);

arrTargetIPAddr := F_ScanIPv4AddrIds(strTargetIPAddr);
nSyncOffset := arrTargetIPAddr[3] MOD 10;

nSyncOffset_1		:= nSyncOffset * TIME_TO_DINT(tTaskTime);

sString_1 := '_1st_RGST$07$04;$02CT=11;DS=HTTPS://Y2WM.CN/99.1000.1/AC12bTPL1003RC78N3TRBUQME1J4XR9ZC;OG=0;QS=1;UE=1.00;XP=19;YP=-5;AP=91;CS=05.6;SC=0056;PN=1;$03$04';
sString_2 := '_2nd_RGST$07$04;$02CT=11;DS=HTTPS://Y2WM.CN/99.1000.1/AC12bTPL1003RC78N3TRBUQME1J4XR9ZC;OG=0;QS=1;UE=1.00;XP=19;YP=-5;AP=91;CS=05.6;SC=0056;PN=1;$03$04';

bConcuted := CONCAT2(pSrcString1 := ADR(sString_1), pSrcString2 := ADR(sString_2), pDstString := ADR(sConcuted), SIZEOF(sConcuted));

nSize_1 := LEN(sString_1);
nSize_2 := LEN(sString_2);
nSize_3 := LEN2(ADR(sConcuted));

nStatusByte := ASC(MID(sString_1, nBytesQuantity, bitNO));
nStatusByte.0;
nStatusByte.1;
nStatusByte.2;
nStatusByte.3;
nStatusByte.4;
nStatusByte.5;
nStatusByte.6;
nStatusByte.7;

sString_4	:= MID(sString_1, 4, 6);

//strTCPRxDebug[1] := sStringTest;

FOR nIndex := 1 TO 20 DO
	strTCPRxDebug[nIndex] := CONCAT(CONCAT('_MESSAGE_NO_', INT_TO_STRING(nIndex)), '_'); 	
END_FOR

nSizeTCPRxDebug 	:= SIZEOF(strTCPRxDebug);
nSizeTCPRxDebug_1	:= SIZEOF(strTCPRxDebug[1]);

MEMMOVE(ADR(strTCPRxDebug[2]), ADR(strTCPRxDebug[1]), SIZEOF(strTCPRxDebug)-SIZEOF(strTCPRxDebug[1]));

END_PROGRAM
